DATA_BLOCK "ID_Plate_CM_DI_iPlateSenNotBlack"
{ S7_Optimized_Access := 'FALSE' }
VERSION : 0.1
NON_RETAIN
"FB_CM_DI_Sensor"

BEGIN

END_DATA_BLOCK

